// TwinCAT 3 PLC project PLC_PFRJ
// ProgramVersion: 3.1.4024.0
// libraries:
//   Tc2_Standard, * (Beckhoff Automation GmbH)
//   Tc2_System, * (Beckhoff Automation GmbH)
//   Tc2_Utilities, * (Beckhoff Automation GmbH)
//   Tc3_IoLink, * (Beckhoff Automation GmbH)
//   Tc3_Module, * (Beckhoff Automation GmbH)
//   VisuDialogs, * (System)
//   VisuSymbols,3.5.10.0,System
// project tree:
//   / DataCollectionTask.TcTTO, GlobalTextList.TcGTLO, PlcTask.TcTTO, Visualization Manager.TcVMO (not stored)
//   GVLs/ gIO.TcGVL, gMachine.TcGVL, gMachineSettings.TcGVL, gScaledIO.TcGVL, gHMI.TcGVL
//   POUs/DataCollection/ MonitoredValue.TcDUT, MonitoredValueUpdate.TcPOU, ScaledValue.TcPOU
//   POUs/HMI/ HMI_FB.TcPOU
//   POUs/ MAIN_ST.TcDUT, MAIN.TcPOU
//   POUs/TestCell/ TEST_STATE.TcDUT, TestFB.TcPOU, SafetyParameters.TcDUT, TestCell.TcDUT, TestParameters.TcDUT
//   POUs/UtilityFunctions/ TSIG.TcPOU
//   VISUs/ Visualization.TcVIS
// real-time tasks:
//   TASK PlcTask: cycle T#10ms, priority 20, ADS port 350
//   TASK DataCollectionTask: cycle T#10ms, priority 1, ADS port 351
// I/O:
//   DEVICE Device 1 (Beckhoff CCAT)
//   DEVICE Device 2 (EtherCAT), AmsNetId 5.131.46.11.3.1
//     Term 1 (EK1200) [EK1200-5000 EtherCAT Power supply (2A E-Bus)]
//       Term 2 (EL2124) [EL2124 4Ch. Dig. Output 5V, 20mA]
//       Term 3 (EL1018) [EL1018 8Ch. Dig. Input 24V, 10µs]
//       Term 4 (EL2008) [EL2008 8Ch. Dig. Output 24V, 0.5A]
//       Term 5 (EL2008) [EL2008 8Ch. Dig. Output 24V, 0.5A]
//       Term 6 (EL2008) [EL2008 8Ch. Dig. Output 24V, 0.5A]
//       Term 7 (EL3068) [EL3068 8Ch. Ana. Input 0-10V]
//       Term 8 (EL3318) [EL3318 8Ch. Ana Input Thermocouple (TC)]
//       Term 9 (EK1122) [EK1122 2 port EtherCAT junction]
//       Term 10 (EL9011) [EL9011 End Terminal]
// variable links:
//   PLC_PFRJ/PLC_PFRJ Instance <-> Device 2 (EtherCAT)/Term 1 (EK1200)/Term 2 (EL2124)
//     PlcTask Outputs/gIO.DO_CollectData <-> Channel 3/Output
//     PlcTask Outputs/gIO.DO_ZVSIgnite <-> Channel 1/Output
//   PLC_PFRJ/PLC_PFRJ Instance <-> Device 2 (EtherCAT)/Term 1 (EK1200)/Term 3 (EL1018)
//     PlcTask Inputs/gIO.DI_24VAtSolenoids <-> Channel 3/Input
//     PlcTask Inputs/gIO.DI_ESTOP_L1 <-> Channel 5/Input
//     PlcTask Inputs/gIO.DI_ESTOP_L2 <-> Channel 6/Input
//   PLC_PFRJ/PLC_PFRJ Instance <-> Device 2 (EtherCAT)/Term 1 (EK1200)/Term 4 (EL2008)
//     PlcTask Outputs/gIO.DO_CombustorAirSolenoid <-> Channel 2/Output
//     PlcTask Outputs/gIO.DO_EjectorSolenoid <-> Channel 8/Output
//     PlcTask Outputs/gIO.DO_MethaneSolenoid <-> Channel 3/Output
//     PlcTask Outputs/gIO.DO_SeederExtendSolenoid <-> Channel 6/Output
//     PlcTask Outputs/gIO.DO_SeederFluidization <-> Channel 7/Output
//     PlcTask Outputs/gIO.DO_SeederRetractSolenoid <-> Channel 5/Output
//     PlcTask Outputs/gIO.DO_WaterQuenchSolenoid <-> Channel 4/Output
//   PLC_PFRJ/PLC_PFRJ Instance <-> Device 2 (EtherCAT)/Term 1 (EK1200)/Term 6 (EL2008)
//     PlcTask Outputs/gIO.DO_Reset <-> Channel 5/Output
//   PLC_PFRJ/PLC_PFRJ Instance <-> Device 2 (EtherCAT)/Term 1 (EK1200)/Term 7 (EL3068)
//     PlcTask Inputs/gIO.AI_AirInletPressure <-> AI Standard Channel 1/Value
//     PlcTask Inputs/gIO.AI_CombustorPressure <-> AI Standard Channel 7/Value
//     PlcTask Inputs/gIO.AI_EjectorPressure <-> AI Standard Channel 3/Value
//     PlcTask Inputs/gIO.AI_ExtendPressure <-> AI Standard Channel 6/Value
//     PlcTask Inputs/gIO.AI_FacilityPressure <-> AI Standard Channel 4/Value
//     PlcTask Inputs/gIO.AI_FluidizationPressure <-> AI Standard Channel 5/Value
//     PlcTask Inputs/gIO.AI_LoadCellWeight <-> AI Standard Channel 8/Value
//     PlcTask Inputs/gIO.AI_MethaneInletPressure <-> AI Standard Channel 2/Value

CONFIGURATION PLC_PFRJ
    RESOURCE PLC ON TwinCAT3
        TASK DataCollectionTask(INTERVAL := T#10ms, PRIORITY := 1);
        TASK PlcTask(INTERVAL := T#10ms, PRIORITY := 20);
        PROGRAM MAIN WITH PlcTask : MAIN;
    END_RESOURCE
END_CONFIGURATION

// ---- POUs/DataCollection/MonitoredValue.TcDUT
TYPE MonitoredValue :
STRUCT
	rawValue          : INT;
	rawValueMin       : INT;
	rawValueMax       : INT;
	scaledValue       : REAL;
	scaledValueMin    : REAL;
	scaledValueMax    : REAL;
	units             : STRING(10);
	lowerWarningValue : REAL;
	upperWarningValue : REAL; 
	dbName            : STRING(50);
END_STRUCT
END_TYPE

// ---- POUs/MAIN_ST.TcDUT
{attribute 'qualified_only'}
{attribute 'strict'}
TYPE MAIN_ST :
(
	STARTUP,
	IDLE,
	TESTING,
	ESTOP,
	WAIT_FOR_RESET,
	RESETTING
);
END_TYPE

// ---- POUs/TestCell/TEST_STATE.TcDUT
{attribute 'qualified_only'}
{attribute 'strict'}
TYPE TEST_STATE :
(
	STARTUP,
	IDLE,
	CHECK_TEST_READY,
	SET_TEST_VARIABLES,
	START_TEST,
	START_IGNITION,
	CHECK_IGNITION,
	WAIT_FOR_SEED,
	RUN_TEST,
	ERROR,
	COMPLETE,
	START_BLOWDOWN,
	BLOWDOWN,
	BLOWDOWN_COMPLETE,
	STOP,
	ESTOP,
	WAIT_FOR_RESET,
	RESETTING
);
END_TYPE

// ---- POUs/TestCell/SafetyParameters.TcDUT
TYPE SafetyParameters :
STRUCT
	minAirPressure          : REAL := 30;
	maxAirPressureDelay     : TIME := T#2S;
	minFacilityPressure     : REAL := 150;
	minMethanePressure      : REAL := 20;
	maxMethanePressureDelay : TIME := T#1S;
	minCombustorPressure    : REAL;
	minIgnitionDelay        : TIME := T#1S;
	
	bOverrideMethaneCheck      : BOOL := FALSE;
	bOverrideFacilityAirCheck  : BOOL := FALSE;
	bOverrideIngitionCheck     : BOOL := FALSE;
END_STRUCT
END_TYPE

// ---- POUs/TestCell/TestCell.TcDUT
TYPE TestCell :
STRUCT
	//Watchdog timers
	fbTON_TestTimer              :  TON;
	fbTON_AirAtPressure          :  TON;
	fbTon_ZVSTimer               :  TON;
	fbTon_MethaneTimer           :  TON;
	fbTon_SeedTime               :  TON;
	fbTon_PistonDelay            :  TON;
	fbTon_PowderIgnitionDelay	 :  TON;
	fbTon_EjectorDelay           :  TON;
	fbTon_ZVSTrigger             :  TON;
	
	//Test Signals and Pulse Generators
	TSIG_ZVSIgnite               :  TSIG;
	TSIG_CombustorAirSolenoid    :  TSIG;
	TSIG_MethaneSolenoid         :  TSIG;
	TSIG_WaterQuenchSolenoid     :  TSIG;
	TSIG_SeederExtendSolenoid    :  TSIG;
	TSIG_SeederRetractSolenoid   :  TSIG;
	TSIG_FluidizationSolenoid    :  TSIG;
	TSIG_EjectorSolenoid         :  TSIG;
	
	//MAIN PROGRAM STATE MACHINE
	state : TEST_STATE := TEST_STATE.STARTUP;
	
	//HMI_Commands
	command_StartTest : BOOL;
	command_StopTest  : BOOL;
	command_Reset     : BOOL;
	command_RunSeed   : BOOL := FALSE;
	
	//test variables
	testComplete     : BOOL;
	testTime         : TIME;
	airPressureTime  : TIME := T#2S;

END_STRUCT
END_TYPE

// ---- POUs/TestCell/TestParameters.TcDUT
TYPE TestParameters :
STRUCT
	ZVSIgniteOnTime					: TIME := T#10S;
	ZVSIgniteOffTime				: TIME := T#12S;
	CombustorAirSolenoidOnTime		: TIME := T#0S;       
	CombustorAirSolenoidOffTime		: TIME := T#25S;
	MethaneSolenoidOnTime			: TIME := T#0S;
	MethaneSolenoidOffTime			: TIME := T#0S; 
	WaterQuenchSolenoidOnTime 		: TIME := T#0S;
	WaterQuenchSolenoidOffTime		: TIME := T#0S;
	SeederExtendSolenoidOnTime		: TIME := T#0S;
	SeederExtendSolenoidOffTime		: TIME := T#0S;
	SeederRetractSolenoidOnTime		: TIME := T#0S;
	SeederRetractSolenoidOffTime	: TIME := T#0S;
	FluidizationSolenoidOnTime		: TIME := T#0S;
	FluidizationSolenoidOffTime		: TIME := T#0S;
	EjectorSolenoidOnTime           : TIME := T#0S;
	EjectorSolenoidOffTime          : TIME := T#0S;
	
END_STRUCT
END_TYPE

// ---- GVLs/gIO.TcGVL
{attribute 'qualified_only'}
VAR_GLOBAL
	
	//Digital Outputs
	DO_ZVSIgnite             AT %Q* : BOOL;
	DO_CombustorAirSolenoid  AT %Q* : BOOL;
	DO_MethaneSolenoid       AT %Q* : BOOL;
	DO_WaterQuenchSolenoid   AT %Q* : BOOL;  
	DO_SeederExtendSolenoid  AT %Q* : BOOL;	
	DO_SeederRetractSolenoid AT %Q* : BOOL;
	DO_SeederFluidization    AT %Q* : BOOL;
	DO_Reset                 AT %Q* : BOOL;
	DO_CollectData           AT %Q* : BOOL;
	DO_EjectorSolenoid       AT %Q* : BOOL;
	
	//Digital Inputs
	DI_SeederExtendLimitSensor  AT %I* : BOOL;
	DI_SeederRetractLimitSensor AT %I* : BOOL;
	DI_MotorExtendLimitSensor   AT %I* : BOOL;
	DI_MotorRetractLimitSensor  AT %I* : BOOL;  
	DI_24VAtSolenoids           AT %I* : BOOL;
	DI_ESTOP_L1                 AT %I* : BOOL;
	DI_ESTOP_L2                 AT %I* : BOOL;
	
	//AnalogInputs
	AI_CombustorPressure        AT %I* : INT;
	AI_AirInletPressure         AT %I* : INT;
	AI_MethaneInletPressure     AT %I* : INT;
	AI_FacilityPressure         AT %I* : INT;
	AI_CombustorLightIntensity  AT %I* : INT;
	AI_FluidizationPressure     AT %I* : INT;
	AI_EjectorPressure          AT %I* : INT;
	AI_LoadCellWeight           AT %I* : INT;
	AI_ExtendPressure           AT %I* : INT;
	TC_CombustorTemperature     AT %I* : INT;
	
	
	//Analog Outputs
	AO_FluidizationValvePos     AT %Q* : INT;
	
	
END_VAR

// ---- GVLs/gMachine.TcGVL
{attribute 'qualified_only'}
VAR_GLOBAL
	testCell : TestCell;
END_VAR

// ---- GVLs/gMachineSettings.TcGVL
{attribute 'qualified_only'}
VAR_GLOBAL
	
	safetyParameters : SafetyParameters;
	testParameters   : TestParameters;
	
	
	//Communications
	temperatureThreshold  : REAL;
	IoLinkAmsId           : ARRAY[0..5] OF BYTE := [5,131,46,11,3,14];
	IoLinkPort            : UINT := E_IolPort.Port1;	
	
	//testVariables
	motorSeederActive     : BOOL;
	pistonSeederActive    : BOOL;
	
END_VAR

// ---- GVLs/gScaledIO.TcGVL
{attribute 'qualified_only'}
VAR_GLOBAL
	monitoredValues : ARRAY[0..16] OF MonitoredValue;
END_VAR

// ---- GVLs/gHMI.TcGVL
{attribute 'qualified_only'}
VAR_GLOBAL
	//HMI BUTTONS
	bStartButtonState            : BOOL;
	bStopButtonState             : BOOL;
	bStartSeedButton			 : BOOL;
	bAirSolenoidButton           : BOOL;
	bFuelSolenoidButton          : BOOL;
	bWaterQuenchSolenoidButton   : BOOL;
	bZVSSolenoidButton           : BOOL;
	bFluidizationSolenoidButton  : BOOL;
	bSeederExtendSolenoidButton  : BOOL;
	bSeederRetractSolenoidButton : BOOL;
	bQDCMethaneSolenoidButton    : BOOL;
	bReset                       : BOOL;
	
	//HMI DATA FIELDS
	iAirStartTime                : INT;
	iAirStopTime                 : INT;
	iFuelStartTime               : INT;
	iFuelStopTime                : INT;
	iWaterQuenchStartTime        : INT;
	iWaterQuenchStopTime         : INT; 
	iZVSStartTime                : INT;
	iZVSStopTime                 : INT;
	iFluidizationStartTime       : INT;
	iFluidizationStopTime        : INT;
	iSeederExtendStartTime       : INT;
	iSeederExtendStopTime        : INT;
	iSeederRetractStartTime      : INT;
	iSeederRetractStopTime       : INT;
	iQDCMethaneStartTime         : INT;
	iQDCMethaneStopTime          : INT;
	
	//HMI User Feedback
	iBlowdownTimeProgress        : INT;
	bEStopPressed                : BOOL;
	seedTime                     : STRING(16);
	
END_VAR

// ---- POUs/MAIN.TcPOU
PROGRAM MAIN
VAR
	testFB : TestFB;
	monitoredValueUpdate : MonitoredValueUpdate;
	main_state : MAIN_ST := MAIN_ST.STARTUP;
	hmi_FB   : HMI_FB;
	
	//main variables 
	bInputError : BOOL := FALSE;
END_VAR

//Always run the function blocks
testFB();
monitoredValueUpdate();
hmi_FB();

IF NOT gIO.DI_ESTOP_L2 THEN
	main_state := MAIN_ST.ESTOP;
END_IF

CASE MAIN_STATE OF 
	MAIN_ST.STARTUP: 
		testFB(command_StartTest:=FALSE, command_StopTest:=FALSE,command_Reset:=FALSE);
		monitoredValueUpdate(resetDefaults:=TRUE);
		main_state := MAIN_ST.IDLE;
	MAIN_ST.IDLE:
		IF gHMI.bStartButtonState THEN
			gHMI.bStartButtonState := FALSE;
			main_state := MAIN_ST.TESTING;
			testFB(command_StartTest:=TRUE, bNoMethane:=NOT gHMI.bMethaneCheckBox);
		END_IF
	MAIN_ST.TESTING:
		IF gHMI.bStopButtonState THEN
			gHMI.bStopButtonState := FALSE;
			testFB(command_StopTest:=TRUE);
		END_IF
		IF gHMI.bStartSeedButtonState AND NOT testFB.bSeedInhibit THEN
			gHMI.bStartSeedButtonState := FALSE;
			testFB(command_StartSeed := TRUE);
		END_IF
		IF gMachine.testCell.state = TEST_STATE.COMPLETE 
			OR gMachine.testCell.state = TEST_STATE.STOP
			OR gMachine.testCell.state = TEST_STATE.ESTOP THEN
				main_state := MAIN_ST.IDLE;
		END_IF
	MAIN_ST.ESTOP:
		gMachine.testCell.state := TEST_STATE.ESTOP;
		IF gIO.DI_ESTOP_L2 THEN
			gMachine.testCell.state := TEST_STATE.WAIT_FOR_RESET;
			main_state := MAIN_ST.WAIT_FOR_RESET;
			
		END_IF
	MAIN_ST.WAIT_FOR_RESET:
		IF gHMI.bReset THEN
			gHMI.bReset := FALSE;
			testFB(command_Reset:=TRUE);
			main_state := MAIN_ST.RESETTING;
		END_IF
	MAIN_ST.RESETTING:
		IF gMachine.testCell.state = TEST_STATE.IDLE THEN
			main_state := MAIN_ST.IDLE;
		END_IF	
END_CASE

gHMI.bEStopPressed := NOT gIO.DI_24VAtSolenoids;

END_PROGRAM

// ---- POUs/TestCell/TestFB.TcPOU
FUNCTION_BLOCK TestFB
VAR_INPUT
	//Test inputs
	command_StartTest : BOOL;
	command_StopTest  : BOOL;
	command_Reset     : BOOL;
	command_StartSeed : BOOL;
END_VAR
VAR_OUTPUT
	errorDiagMsg		: STRING(255);
	bStartSeedInhibit        : BOOL := FALSE;
	bTestInhibit		: BOOL := FALSE;
END_VAR
VAR
	bStartup          : BOOL  := TRUE;
	methaneStartUpDelay		: TON;
	methaneSettingTime		: TON;
	ignitionTimer       	: TON;
	ignitionDelay 			: TON;
	ignitionCheckTimer		: TON;
	testTimer				: TON;
END_VAR

IF command_StopTest THEN
	command_StopTest := FALSE;
	gMachine.testCell.state := TEST_STATE.STOP;
END_IF

//Use inhibits
bStartSeedInhibit := NOT (gMachine.testCell.state = TEST_STATE.WAIT_FOR_SEED);

CASE gMachine.testCell.state OF
	TEST_STATE.STARTUP:
		IF bStartup THEN
			bStartup := FALSE;
			gMachine.testCell.TSIG_ZVSIgnite(Init:=FALSE, pIO:=ADR(gIO.DO_ZVSIgnite));
			gMachine.testCell.TSIG_CombustorAirSolenoid(Init:=FALSE, pIO:=ADR(gIO.DO_CombustorAirSolenoid));   
			gMachine.testCell.TSIG_MethaneSolenoid(Init:=FALSE, pIO:=ADR(gIO.DO_MethaneSolenoid));      
			gMachine.testCell.TSIG_WaterQuenchSolenoid(Init:=FALSE, pIO:=ADR(gIO.DO_WaterQuenchSolenoid));  
			gMachine.testCell.TSIG_SeederExtendSolenoid(Init:=FALSE, pIO:=ADR(gIO.DO_SeederExtendSolenoid));    
			gMachine.testCell.TSIG_SeederRetractSolenoid(Init:=FALSE, pIO:=ADR(gIO.DO_SeederRetractSolenoid));  
			gMachine.testCell.TSIG_FluidizationSolenoid(Init:=FALSE, pIO:=ADR(gIO.DO_SeederFluidization));   
			gMachine.testCell.TSIG_EjectorSolenoid(Init:=FALSE, pIO:=ADR(gIO.DO_EjectorSolenoid));     
			gMachine.testCell.state := TEST_STATE.IDLE;	
		END_IF
		
	TEST_STATE.IDLE:
		//Make sure all timers are reset from the idle state
		IF command_StartTest THEN
			command_StartTest := FALSE;
			gMachine.testCell.state := TEST_STATE.CHECK_TEST_READY;
		END_IF
		
	TEST_STATE.CHECK_TEST_READY:
		gMachine.testCell.state := TEST_STATE.SET_TEST_VARIABLES;
		
	TEST_STATE.SET_TEST_VARIABLES:
		gMachine.testCell.state := TEST_STATE.START_TEST;
	TEST_STATE.START_TEST:
		gIO.DO_CollectData := TRUE;
		gIO.DO_CombustorAirSolenoid := TRUE;
		methaneStartUpDelay(IN:=TRUE, PT:=T#2S);
		IF methaneStartUpDelay.Q THEN
			IF gScaledIO.monitoredValues[1].scaledValue > gMachineSettings.safetyParameters.minAirPressure THEN
				methaneStartUpDelay(IN:=FALSE);
				gIO.DO_MethaneSolenoid := TRUE;
				gMachine.testCell.state := TEST_STATE.START_IGNITION;
			ELSE
				methaneStartUpDelay(IN:=FALSE);
				errorDiagMsg := 'Methane flow attempted without air';
				gMachine.testCell.state := TEST_STATE.ERROR;
			END_IF
		END_IF
	
	TEST_STATE.START_IGNITION:
		ignitionDelay(IN:=TRUE, PT:=T#1S);
		IF ignitionDelay.Q THEN
			IF gScaledIO.monitoredValues[2].scaledValue > gMachineSettings.safetyParameters.minMethanePressure THEN 
				gIO.DO_ZVSIgnite := TRUE;
				ignitionTimer(IN:=TRUE, PT:=T#4S);
				IF ignitionTimer.Q THEN
					gIO.DO_ZVSIgnite := FALSE;
					ignitionDelay(IN:=FALSE);
					ignitionTimer(IN:=FALSE);
					gMachine.testCell.state := TEST_STATE.CHECK_IGNITION;
				END_IF
			ELSE
				ignitionDelay(IN:=FALSE);
				ignitionTimer(IN:=FALSE);
				errorDiagMsg := 'Ignition Attempted Without Methane';
				gMachine.testCell.state := TEST_STATE.ERROR;	
			END_IF
		END_IF
		
	TEST_STATE.CHECK_IGNITION: 
		ignitionCheckTimer(IN:=TRUE, PT:=T#0.25S);
		IF ignitionCheckTimer.Q THEN
			ignitionCheckTimer(IN:=FALSE);
			IF gScaledIO.monitoredValues[7].scaledValue > gMachineSettings.safetyParameters.minCombustorPressure THEN
				gMachine.testCell.state := TEST_STATE.WAIT_FOR_SEED;	
			ELSE
				errorDiagMsg := 'Ignition failure, no combustion occured';
				gMachine.testCell.state := TEST_STATE.ERROR;	
			END_IF
		END_IF
	
	TEST_STATE.WAIT_FOR_SEED:
		IF command_StartSeed THEN
			gMachine.testCell.state := TEST_STATE.RUN_TEST;
		END_IF
		
	TEST_STATE.RUN_TEST:
		//Start time based systems
		testTimer(IN:=TRUE, PT:=MAX(gMachineSettings.testParameters.ZVSIgniteOffTime, 
									gMachineSettings.testParameters.MethaneSolenoidOffTime, 
									gMachineSettings.testParameters.SeederExtendSolenoidOffTime, 
									gMachineSettings.testParameters.FluidizationSolenoidOffTime));
		gIO.DO_EjectorSolenoid := TRUE;
		gMachine.testCell.TSIG_ZVSIgnite(Init:=TRUE, Start_Time:=gMachineSettings.testParameters.ZVSIgniteOnTime,End_Time:=gMachineSettings.testParameters.ZVSIgniteOffTime);
		gMachine.testCell.TSIG_MethaneSolenoid(Init:=TRUE, Start_Time:=gMachineSettings.testParameters.MethaneSolenoidOnTime, End_Time:=gMachineSettings.testParameters.MethaneSolenoidOffTime);
		gMachine.testCell.TSIG_SeederExtendSolenoid(Init:=TRUE, Start_Time:=gMachineSettings.testParameters.SeederExtendSolenoidOnTime, End_Time:=gMachineSettings.testParameters.SeederExtendSolenoidOffTime);
		gMachine.testCell.TSIG_FluidizationSolenoid(Init:=TRUE, Start_Time:=gMachineSettings.testParameters.FluidizationSolenoidOnTime, End_Time:=gMachineSettings.testParameters.FluidizationSolenoidOffTime);
	
		//run watchdog tests
		//IF gIO.DI_SeederExtendLimitSensor THEN
		//	testTimer(IN:=FALSE);
		//	gMachine.testCell.state := TEST_STATE.COMPLETE;
		//END_IF
		IF 	testTimer.Q THEN
			testTimer(IN:=FALSE);
			gMachine.testCell.state := TEST_STATE.COMPLETE;
		END_IF
		IF  gScaledIO.monitoredValues[1].scaledValue < gMachineSettings.safetyParameters.minAirPressure THEN
			errorDiagMsg := 'Loss of air pressure during testing'; 
			gMachine.testCell.state := TEST_STATE.ERROR;
		END_IF
		
		IF 	gScaledIO.monitoredValues[2].scaledValue < gMachineSettings.safetyParameters.minMethanePressure THEN
			errorDiagMsg := 'Loss of methane pressure during testing'; 
			gMachine.testCell.state := TEST_STATE.ERROR;
		END_IF
		
		IF 	gScaledIO.monitoredValues[7].scaledValue < gMachineSettings.safetyParameters.minCombustorPressure THEN
			errorDiagMsg := 'Loss of chamber pressure, unstarted engine';
			gMachine.testCell.state := TEST_STATE.ERROR;
		END_IF
		
		IF gScaledIO.monitoredValues[4].scaledValue < gMachineSettings.safetyParameters.minFacilityPressure THEN
			errorDiagMsg := 'Tank pressure too low during testing';
			gMachine.testCell.state := TEST_STATE.ERROR;
		END_IF
		
	TEST_STATE.COMPLETE:
		//reset timers
		gMachine.testCell.TSIG_ZVSIgnite(Init:=FALSE);
		gMachine.testCell.TSIG_CombustorAirSolenoid(Init:=FALSE);   
		gMachine.testCell.TSIG_MethaneSolenoid(Init:=FALSE);      
		gMachine.testCell.TSIG_WaterQuenchSolenoid(Init:=FALSE);  
		gMachine.testCell.TSIG_SeederExtendSolenoid(Init:=FALSE);    
		gMachine.testCell.TSIG_SeederRetractSolenoid(Init:=FALSE);  
		gMachine.testCell.TSIG_FluidizationSolenoid(Init:=FALSE);   
		gMachine.testCell.TSIG_EjectorSolenoid(Init:=FALSE);  
		//reset IO
		gIO.DO_CombustorAirSolenoid := FALSE;
		gIO.DO_MethaneSolenoid := FALSE;
		gIO.DO_SeederExtendSolenoid := FALSE;
		gIO.DO_SeederFluidization := FALSE;
		gIO.DO_WaterQuenchSolenoid := FALSE;
		gIO.DO_ZVSIgnite := FALSE;
		gIO.DO_EjectorSolenoid := FALSE;   
		//Go to blowdown post test
		gMachine.testCell.state := TEST_STATE.BLOWDOWN;
	
	TEST_STATE.STOP:
		//reset timers
		gMachine.testCell.TSIG_ZVSIgnite(Init:=FALSE);
		gMachine.testCell.TSIG_CombustorAirSolenoid(Init:=FALSE);   
		gMachine.testCell.TSIG_MethaneSolenoid(Init:=FALSE);      
		gMachine.testCell.TSIG_WaterQuenchSolenoid(Init:=FALSE);  
		gMachine.testCell.TSIG_SeederExtendSolenoid(Init:=FALSE);    
		gMachine.testCell.TSIG_SeederRetractSolenoid(Init:=FALSE);  
		gMachine.testCell.TSIG_FluidizationSolenoid(Init:=FALSE);   
		gMachine.testCell.TSIG_EjectorSolenoid(Init:=FALSE);     
		gMachine.testCell.state := TEST_STATE.BLOWDOWN;
		//run purge air 
	TEST_STATE.BLOWDOWN:
		gMachine.testCell.TSIG_CombustorAirSolenoid(Init:=TRUE, Start_Time := INT_TO_TIME(0), End_Time := INT_TO_TIME(5000));
		gHMI.iBlowdownTimeProgress := REAL_TO_INT(TIME_TO_INT(gMachine.testCell.TSIG_CombustorAirSolenoid.ET - gMachine.testCell.TSIG_CombustorAirSolenoid.Start_Time) * (100) / TIME_TO_INT(gMachine.testCell.TSIG_CombustorAirSolenoid.End_Time - gMachine.testCell.TSIG_CombustorAirSolenoid.Start_Time));
		IF NOT gMachine.testCell.TSIG_CombustorAirSolenoid.Q THEN
			gMachine.testCell.state := TEST_STATE.BLOWDOWN_COMPLETE;
		END_IF
	TEST_STATE.BLOWDOWN_COMPLETE:
		gMachine.testCell.TSIG_CombustorAirSolenoid(Init:=FALSE);
		gHMI.iBlowdownTimeProgress := 0;
		gMachine.testCell.state := TEST_STATE.IDLE;
		
	TEST_STATE.ESTOP: 
		gMachine.testCell.TSIG_ZVSIgnite(Init:=FALSE);
		gMachine.testCell.TSIG_CombustorAirSolenoid(Init:=FALSE);   
		gMachine.testCell.TSIG_MethaneSolenoid(Init:=FALSE);      
		gMachine.testCell.TSIG_WaterQuenchSolenoid(Init:=FALSE);  
		gMachine.testCell.TSIG_SeederExtendSolenoid(Init:=FALSE);    
		gMachine.testCell.TSIG_SeederRetractSolenoid(Init:=FALSE);  
		gMachine.testCell.TSIG_FluidizationSolenoid(Init:=FALSE);   
		gMachine.testCell.TSIG_EjectorSolenoid(Init:=FALSE);    
		
		//reset IO
		gIO.DO_CombustorAirSolenoid := FALSE;
		gIO.DO_MethaneSolenoid := FALSE;
		gIO.DO_SeederExtendSolenoid := FALSE;
		gIO.DO_SeederFluidization := FALSE;
		gIO.DO_WaterQuenchSolenoid := FALSE;
		gIO.DO_ZVSIgnite := FALSE;
		gIO.DO_EjectorSolenoid := FALSE;
	
			
	TEST_STATE.WAIT_FOR_RESET:
		IF command_Reset THEN
			command_Reset := FALSE;
			gIO.DO_Reset  := TRUE;
			gMachine.testCell.state := TEST_STATE.RESETTING;
		END_IF
		
	TEST_STATE.RESETTING: 
		IF gIO.DI_24VAtSolenoids THEN
			gIO.DO_Reset := FALSE;
			gMachine.testCell.state := TEST_STATE.IDLE;
		END_IF	
	
	TEST_STATE.ERROR: 
		gMachine.testCell.state := TEST_STATE.STOP;
		
END_CASE

END_FUNCTION_BLOCK

// ---- POUs/DataCollection/ScaledValue.TcPOU
FUNCTION ScaledValue : REAL
VAR_INPUT
	mv : MonitoredValue;
END_VAR
VAR
END_VAR

IF (mv.rawValueMax - mv.rawValueMin) > 0 THEN
	ScaledValue := mv.scaledValueMin + (mv.rawValue - mv.rawValueMin) * ((mv.scaledValueMax- mv.scaledValueMin) / (mv.rawValueMax - mv.rawValueMin));
END_IF

END_FUNCTION

// ---- POUs/DataCollection/MonitoredValueUpdate.TcPOU
FUNCTION_BLOCK MonitoredValueUpdate
VAR_INPUT
	resetDefaults : BOOL := TRUE;
END_VAR
VAR_OUTPUT
END_VAR
VAR
	//Declare the array of monitored values
	monitoredValues : ARRAY[0..16] OF MonitoredValue;
END_VAR

IF resetDefaults THEN
	resetDefaults := FALSE;
	//Pressure Transducers
	monitoredValues[1].rawValueMin       := 0;
	monitoredValues[1].rawValueMax       := 32767; 
	monitoredValues[1].scaledValueMin    := 0;
	monitoredValues[1].scaledValueMax    := 200;
	monitoredValues[1].units             := 'psig';
	monitoredValues[1].lowerWarningValue := 0;
	monitoredValues[1].upperWarningValue := 180;
	monitoredValues[1].dbName            := 'air inlet pressure';
	
	monitoredValues[2].rawValueMin       := 0;
	monitoredValues[2].rawValueMax       := 32767; 
	monitoredValues[2].scaledValueMin    := 0;
	monitoredValues[2].scaledValueMax    := 300;
	monitoredValues[2].units             := 'psig';
	monitoredValues[2].lowerWarningValue := 0;
	monitoredValues[2].upperWarningValue := 80;
	monitoredValues[2].dbName            := 'methane inlet pressure';
	
	monitoredValues[3].rawValueMin       := 0;
	monitoredValues[3].rawValueMax       := 32767; 
	monitoredValues[3].scaledValueMin    := -14.7;
	monitoredValues[3].scaledValueMax    := 30;
	monitoredValues[3].units             := 'psig';
	monitoredValues[3].lowerWarningValue := 0;
	monitoredValues[3].upperWarningValue := 30;
	monitoredValues[3].dbName            := 'ejector pressure';
	
	monitoredValues[4].rawValueMin       := 0;
	monitoredValues[4].rawValueMax       := 32767; 
	monitoredValues[4].scaledValueMin    := 0;
	monitoredValues[4].scaledValueMax    := 1000;
	monitoredValues[4].units             := 'psig';
	monitoredValues[4].lowerWarningValue := 150;
	monitoredValues[4].upperWarningValue := 300;
	monitoredValues[4].dbName            := 'facility pressure';
	
	monitoredValues[5].rawValueMin       := 0;
	monitoredValues[5].rawValueMax       := 32767; 
	monitoredValues[5].scaledValueMin    := 0;
	monitoredValues[5].scaledValueMax    := 100;
	monitoredValues[5].units             := 'psig';
	monitoredValues[5].lowerWarningValue := 0;
	monitoredValues[5].upperWarningValue := 15;
	monitoredValues[5].dbName            := 'fluidize pressure';	
	
	monitoredValues[6].rawValueMin       := 0;
	monitoredValues[6].rawValueMax       := 32767; 
	monitoredValues[6].scaledValueMin    := 0;
	monitoredValues[6].scaledValueMax    := 15;
	monitoredValues[6].units             := 'psig';
	monitoredValues[6].lowerWarningValue := 0;
	monitoredValues[6].upperWarningValue := 15;
	monitoredValues[6].dbName            := 'extend pressure';	
	
	monitoredValues[7].rawValueMin       := 0;
	monitoredValues[7].rawValueMax       := 32767; 
	monitoredValues[7].scaledValueMin    := -14.7;
	monitoredValues[7].scaledValueMax    := 100;
	monitoredValues[7].units             := '';
	monitoredValues[7].lowerWarningValue := 0;
	monitoredValues[7].upperWarningValue := 100;
	monitoredValues[7].dbName            := 'combustor pressure';	
	
	monitoredValues[8].rawValueMin       := 0;
	monitoredValues[8].rawValueMax       := 32767; 
	monitoredValues[8].scaledValueMin    := -50;
	monitoredValues[8].scaledValueMax    := 50;
	monitoredValues[8].units             := 'lbm';
	monitoredValues[8].lowerWarningValue := -50;
	monitoredValues[8].upperWarningValue := 50;
	monitoredValues[8].dbName            := 'load cell';	

	
END_IF  

monitoredValues[1].rawValue := gIO.AI_AirInletPressure;
monitoredValues[1].scaledValue := ScaledValue(monitoredValues[1]);

monitoredValues[2].rawValue := gIO.AI_MethaneInletPressure;
monitoredValues[2].scaledValue := ScaledValue(monitoredValues[2]);

monitoredValues[3].rawValue := gIO.AI_EjectorPressure;
monitoredValues[3].scaledValue := ScaledValue(monitoredValues[3]);

monitoredValues[4].rawValue := gIO.AI_FacilityPressure;
monitoredValues[4].scaledValue := ScaledValue(monitoredValues[4]);

monitoredValues[5].rawValue := gIO.AI_FluidizationPressure;
monitoredValues[5].scaledValue := ScaledValue(monitoredValues[5]);

monitoredValues[6].rawValue := gIO.AI_ExtendPressure;
monitoredValues[6].scaledValue := ScaledValue(monitoredValues[6]);

monitoredValues[7].rawValue := gIO.AI_CombustorPressure;
monitoredValues[7].scaledValue := ScaledValue(monitoredValues[7]);

monitoredValues[8].rawValue := gIO.AI_LoadCellWeight;
monitoredValues[8].scaledValue := ScaledValue(monitoredValues[8]);

gScaledIO.monitoredValues := monitoredValues;

END_FUNCTION_BLOCK

// ---- POUs/HMI/HMI_FB.TcPOU
FUNCTION_BLOCK HMI_FB
VAR_INPUT
END_VAR
VAR_OUTPUT
END_VAR
VAR
END_VAR

//HMI DATA FIELDS
gMachineSettings.testParameters.CombustorAirSolenoidOnTime		:= INT_TO_TIME(gHMI.iAirStartTime);        
gMachineSettings.testParameters.CombustorAirSolenoidOffTime 	:= INT_TO_TIME(gHMI.iAirStopTime);               
gMachineSettings.testParameters.FluidizationSolenoidOnTime		:= INT_TO_TIME(gHMI.iFuelStartTime);             
gMachineSettings.testParameters.FluidizationSolenoidOffTime		:= INT_TO_TIME(gHMI.iFuelStopTime);              
gMachineSettings.testParameters.WaterQuenchSolenoidOnTime		:= INT_TO_TIME(gHMI.iWaterQuenchStartTime);      
gMachineSettings.testParameters.WaterQuenchSolenoidOffTime		:= INT_TO_TIME(gHMI.iWaterQuenchStopTime);    
gMachineSettings.testParameters.ZVSIgniteOnTime					:= INT_TO_TIME(gHMI.iZVSStartTime);          
gMachineSettings.testParameters.ZVSIgniteOffTime				:= INT_TO_TIME(gHMI.iZVSStopTime);               
gMachineSettings.testParameters.FluidizationSolenoidOnTime		:= INT_TO_TIME(gHMI.iFluidizationStartTime);  
gMachineSettings.testParameters.FluidizationSolenoidOffTime		:= INT_TO_TIME(gHMI.iFluidizationStopTime);      
gMachineSettings.testParameters.SeederExtendSolenoidOnTime		:= INT_TO_TIME(gHMI.iSeederExtendStartTime);     
gMachineSettings.testParameters.SeederExtendSolenoidOffTime		:= INT_TO_TIME(gHMI.iSeederExtendStopTime);        
gMachineSettings.testParameters.SeederRetractSolenoidOnTime		:= INT_TO_TIME(gHMI.iSeederRetractStartTime);    
gMachineSettings.testParameters.SeederRetractSolenoidOffTime	:= INT_TO_TIME(gHMI.iSeederRetractStopTime);
gMachineSettings.testParameters.MethaneSolenoidOnTime			:= INT_TO_TIME(gHMI.iFuelStartTime);
gMachineSettings.testParameters.MethaneSolenoidOffTime			:= INT_TO_TIME(gHMI.iFuelStopTime); 

gHMI.bReadyForSeed := gMachine.testCell.state = TEST_STATE.WAIT_FOR_SEED;

END_FUNCTION_BLOCK

// ---- POUs/UtilityFunctions/TSIG.TcPOU
FUNCTION_BLOCK PUBLIC TSIG
VAR_INPUT
	Init        : BOOL;
	pIO         : POINTER TO BOOL;
	Start_Time  : TIME;
	End_Time    : TIME;
END_VAR
VAR_OUTPUT
	Q  : BOOL;
	ET : TIME;
END_VAR
VAR
	TimerOn  : TON;
	TimerOff    : TON;
END_VAR

IF (Init AND ET < (End_time - Start_Time) AND Start_Time < End_Time) THEN
	TimerOn(IN:=TRUE, PT:=Start_Time);
	TimerOff(IN:= TimerOn.Q, PT:= (End_Time - Start_Time));
	pIO^ := TimerOn.Q;
	Q := TimerOn.Q;
	ET := TimerOff.ET;
ELSIF (ET = (End_time - Start_Time) AND Init) THEN
	pIO^ := FALSE;
	Q := FALSE;
ELSIF NOT Init THEN
	TimerOn(IN:=FALSE);
	TimerOff(IN:=FALSE);
	Q := FALSE;
	pIO^ := FALSE;
	ET := T#0S; 
END_IF

END_FUNCTION_BLOCK

// ---- GlobalTextList.TcGTLO
TEXTLIST GlobalTextList
  151 = '%f'
  379 = '%i'
  373 = '%q'
  749 = 'Air'
  394 = 'Air Solenoid'
  849 = 'Blowdown Status'
  297 = 'Combustor Pressure (PSI)'
  44 = 'Combustor Temperature'
  519 = 'Confirm Combustion'
  800 = 'Confirm Seed'
  636 = 'Ejector Solenoid'
  380 = 'End Times'
  943 = 'End Times (ms)'
  729 = 'ESTOP'
  364 = 'Fluidization'
  518 = 'Fuel'
  396 = 'Fuel Solenoid'
  615 = 'I5'
  120 = 'Inlet Pressure (PSI)'
  404 = 'Kill Seed'
  627 = 'Manual Control'
  908 = 'Manual Data Collection'
  591 = 'Manual Inputs'
  927 = 'Manual Toggles'
  513 = 'Methane'
  401 = 'Methane Pressure (PSI)'
  660 = 'Motor Subsystem'
  455 = 'Piston Subsystem'
  683 = 'Pressure: %2.3f psi'
  346 = 'QDC Methane'
  287 = 'Quench Solenoid'
  611 = 'Reset'
  646 = 'Retry Ignition'
  750 = 'Retry Ingnition'
  440 = 'Run Seed'
  284 = 'Seeder Extend'
  118 = 'Seeder Fluidization'
  111 = 'Seeder Retract'
  458 = 'Start Test'
  275 = 'Start Time'
  942 = 'Start Times'
  937 = 'Start Times (ms)'
  599 = 'State Machine State'
  486 = 'STOP'
  958 = 'Stop Test'
  459 = 'Stop Time'
  179 = 'System Error'
  121 = 'Tank Pressure (PSI)'
  356 = 'Test Timer'
  864 = 'Time: %2.3f s'
  351 = 'Time: %s'
  119 = 'Water'
  174 = 'ZFS'
  736 = 'ZFS Trigger'
  58 = 'ZVS'
  507 = 'ZVS Trigger'
  692 = '`'
END_TEXTLIST

// ---- VISUs/Visualization.TcVIS
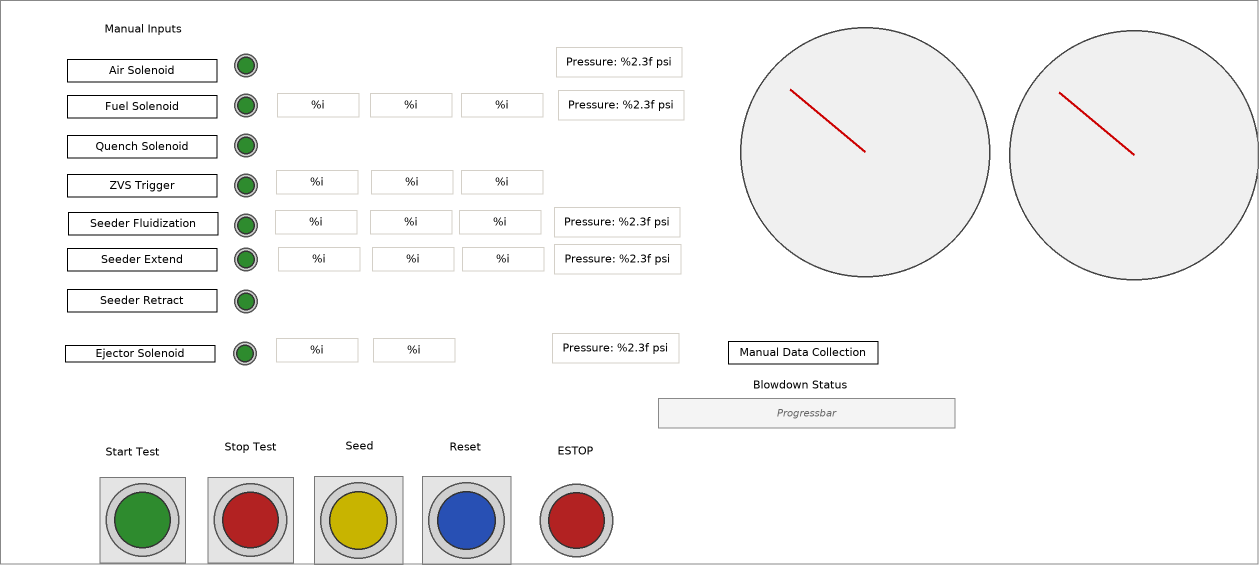
VISUALIZATION Visualization  // 1259x565
    RoundedRectangle (67,59 150x23), "Air Solenoid"
        toggle gIO.DO_CombustorAirSolenoid
    RoundedRectangle (67,95 150x23), "Fuel Solenoid"
        toggle gIO.DO_MethaneSolenoid
    RoundedRectangle (67,135 150x23), "Quench Solenoid"
        toggle gIO.DO_WaterQuenchSolenoid
    RoundedRectangle (67,174 150x23), "ZVS Trigger"
        toggle gIO.DO_ZVSIgnite
    RoundedRectangle (68,212 150x23), "Seeder Fluidization"
        toggle gIO.DO_SeederFluidization
    RoundedRectangle (67,248 150x23), "Seeder Extend"
        toggle gIO.DO_SeederExtendSolenoid
    RoundedRectangle (67,289 150x23), "Seeder Retract"
        toggle gIO.DO_SeederRetractSolenoid
    Label (68,14 150x30), "Manual Inputs"
    Lamp1 (232,52 28x27), variable: gIO.DO_CombustorAirSolenoid, style: Lamp-Lamp1-Green
    Lamp1 (232,92 28x27), variable: gIO.DO_MethaneSolenoid, style: Lamp-Lamp1-Green
    Lamp1 (232,132 28x27), variable: gIO.DO_WaterQuenchSolenoid, style: Lamp-Lamp1-Green
    Lamp1 (232,172 28x27), variable: gIO.DO_ZVSIgnite, style: Lamp-Lamp1-Green
    Lamp1 (232,212 28x27), variable: gIO.DO_SeederFluidization, style: Lamp-Lamp1-Green
    Lamp1 (232,246 28x27), variable: gIO.DO_SeederExtendSolenoid, style: Lamp-Lamp1-Green
    Lamp1 (232,288 28x27), variable: gIO.DO_SeederRetractSolenoid, style: Lamp-Lamp1-Green
    PushSwitch (98,477 89x86), variable: gHMI.bStartButtonState, behaviour: TOGGLE, style: Switch-PushSwitch-Green
    PushSwitch (206,477 89x86), tooltip "STOP", variable: gHMI.bStopButtonState, behaviour: TOGGLE, style: Switch-PushSwitch-Red
    Progressbar (658,398 297x30), variable: gHMI.iBlowdownTimeProgress
    Label (725,370 150x30), "Blowdown Status"
    Label (201,432 99x30), "Stop Test"
    Label (83,437 99x30), "Start Test"
    Lamp1 (532,478 89x85), variable: gHMI.bEStopPressed, style: Lamp-Lamp1-Red
    PushSwitch (422,476 89x89), variable: gHMI.bReset, behaviour: TOGGLE, style: Switch-PushSwitch-Blue
    Label (416,432 99x30), "Reset"
    Label (526,436 99x30), "ESTOP"
    RoundedRectangle (65,345 150x17), "Ejector Solenoid"
        toggle gIO.DO_EjectorSolenoid
    Lamp1 (231,340 28x27), variable: gIO.DO_EjectorSolenoid, style: Lamp-Lamp1-Green
    Textfield (554,207 126x30), "Pressure: %2.3f psi", text variable: MAIN.monitoredValueUpdate.monitoredValues[5].scaledValue
    Textfield (554,244 127x30), "Pressure: %2.3f psi", text variable: MAIN.monitoredValueUpdate.monitoredValues[6].scaledValue
    Textfield (558,90 126x30), "Pressure: %2.3f psi", text variable: MAIN.monitoredValueUpdate.monitoredValues[2].scaledValue
    Textfield (556,47 126x30), "Pressure: %2.3f psi", text variable: MAIN.monitoredValueUpdate.monitoredValues[1].scaledValue
    Textfield (277,93 82x24), "%i", text variable: gHMI.iFuelStartTime
        OnMouseDown: write the text variable via InputWithLimits
    Textfield (370,93 82x24), "%i", text variable: gHMI.iFuelStopTime
        OnMouseDown: write the text variable via InputWithLimits
    Textfield (276,170 82x24), "%i", text variable: gHMI.iZVSStartTime
        OnMouseDown: write the text variable via InputWithLimits, min 0, max 50000
    Textfield (371,170 82x24), "%i", text variable: gHMI.iZVSStopTime
        OnMouseDown: write the text variable via InputWithLimits, min 0, max 50000
    Textfield (370,210 82x24), "%i", text variable: gHMI.iFluidizationStopTime
        OnMouseDown: write the text variable via InputWithLimits, min 0, max 50000
    Textfield (275,210 82x24), "%i", text variable: gHMI.iFluidizationStartTime
        OnMouseDown: write the text variable via InputWithLimits, min 0, max 50000
    Textfield (278,247 82x24), "%i", text variable: gHMI.iSeederExtendStartTime
        OnMouseDown: write the text variable via InputWithLimits, min 0, max 50000
    Textfield (372,247 82x24), "%i", text variable: gHMI.iSeederExtendStopTime
        OnMouseDown: write the text variable via InputWithLimits, min 0, max 50000
    Textfield (276,338 82x24), "%i", text variable: gHMI.iSeederRetractStartTime
        OnMouseDown: write the text variable via InputWithLimits, min 0, max 50000
    Textfield (373,338 82x24), "%i", text variable: gHMI.iSeederRetractStopTime
        OnMouseDown: write the text variable via VisuDialogs.Keypad, min 0, max 50000
    Textfield (552,333 127x30), "Pressure: %2.3f psi", text variable: MAIN.monitoredValueUpdate.monitoredValues[3].scaledValue
    Meter360 (740,27 250x250), value: gScaledIO.monitoredValues[7].scaledValue, style: Meter-Meter360-Gray, scale format: %.1f, scale 0..100
    RoundedRectangle (728,341 150x23), "Manual Data Collection"
        tap gIO.DO_CollectData
    Meter360 (1009,30 250x250), value: gScaledIO.monitoredValues[4].scaledValue, style: Meter-Meter360-Gray, scale format: %.1f, scale 0..300
    Textfield (461,93 82x24), "%i", text variable: gHMI.iFuelStopTime
        OnMouseDown: write the text variable via InputWithLimits
    Textfield (461,170 82x24), "%i", text variable: gHMI.iZVSStopTime
        OnMouseDown: write the text variable via InputWithLimits, min 0, max 50000
    Textfield (459,210 82x24), "%i", text variable: gHMI.iFluidizationStopTime
        OnMouseDown: write the text variable via InputWithLimits, min 0, max 50000
    Textfield (462,247 82x24), "%i", text variable: gHMI.iSeederExtendStopTime
        OnMouseDown: write the text variable via InputWithLimits, min 0, max 50000
    PushSwitch (314,476 89x89), variable: gHMI.bStartSeedButton, behaviour: TOGGLE, style: Switch-PushSwitch-Yellow
    Label (310,431 99x30), "Seed"
END_VISUALIZATION
